(* Logix 5000 project; controller Machine_Maintenance_Lab2 vendor 1 type 14 code 155 rev 36.11; software revision 36.00 *)

TASK MainTask (continuous, watchdog 500 ms) : MainProgram

MODULES
   Local : vendor 1 type 14 code 155 (PointIO 0, rev 36.11)
      Discrete_IO : Embedded (PointIO 1, rev 36.11, Output RPI 20 ms)
END_MODULES

PROGRAM MainProgram   (* main routine TrafficLight *)
VAR
   Clock : FBD_TIMER := (PRE := 1000);
   ClockDone_NSGEWR : BOOL;
   ClockDone_NSREWG : BOOL;
   ClockDone_NSREWY : BOOL;
   ClockDone_NSYEWR : BOOL;
   counter : COUNTER := (PRE := 5);
   CycleCounter : COUNTER := (PRE := 5);
   delay : TIMER := (PRE := 10);
   EmerDone : BOOL;
   Emergency : BOOL;
   HighCycleTimer : COUNTER := (PRE := 700);
   i_CycleDone : ALIAS FOR o_CycleDone;
   i_GreenPB : ALIAS FOR Local:1:I.Data.0;
   i_GreenPB_ConveyorStart : ALIAS FOR i_GreenPB;
   i_GreenPBLight_Conveyor1ON : ALIAS FOR o_GreenPBLight_Conveyor1ON;
   i_NightModeButton : ALIAS FOR Local:1:I.Data.3;
   i_Pause : ALIAS FOR Pause;
   i_Piston : ALIAS FOR Local:1:O.Data.2;
   i_RedPB_StopButton : ALIAS FOR Local:1:I.Data.1;
   i_RedPBLight_Conveyor2ON : ALIAS FOR o_RedPBLight_Conveyor2ON;
   i_Turnkey : ALIAS FOR Local:1:I.Data.2;
   i_Turnkey_ItemSensor : ALIAS FOR i_Turnkey;
   ItemCounter1 : COUNTER := (PRE := 5);
   ItemCounterLeft : COUNTER := (PRE := 5);
   ItemCounterRight : COUNTER := (PRE := 6);
   LowCycleTimer : COUNTER := (PRE := 300);
   MaxState : DINT;
   myClock : FBD_TIMER;
   NewCycle : BOOL;
   NightMode : BOOL;
   o_CycleDone : BOOL;
   o_EWG : ALIAS FOR Local:1:O.Data.15;
   o_EWR : ALIAS FOR Local:1:O.Data.13;
   o_EWY : ALIAS FOR Local:1:O.Data.14;
   o_GreenPBLight : ALIAS FOR Local:1:O.Data.0;
   o_GreenPBLight_Conveyor1ON : ALIAS FOR o_GreenPBLight;
   o_NSG : ALIAS FOR Local:1:O.Data.7;
   o_NSR : ALIAS FOR Local:1:O.Data.5;
   o_NSY : ALIAS FOR Local:1:O.Data.6;
   o_Piston : ALIAS FOR i_Piston;
   o_RedPBLight : ALIAS FOR Local:1:O.Data.1;
   o_RedPBLight_Conveyor2ON : ALIAS FOR o_RedPBLight;
   OS_Out : BOOL;
   Pause : BOOL;
   preStart : DINT;
   resetBit : BOOL;
   ResetDelay : TIMER := (PRE := 500);
   Start : BOOL;
   StateCounter : FBD_COUNTER;
   ThreeSecTimer : TIMER := (PRE := 3000);
   timer : TIMER := (PRE := 5000);
   timerDoneLatch : BOOL;
   TimerHighCycle : TIMER := (PRE := 700);
   TimerLowCycle : TIMER := (PRE := 300);
   timerMem : BOOL;
   timerState : DINT;
   TurnkeyOneShot : BOOL := 1;
END_VAR

ROUTINE TrafficLight   (* structured text *)
   
   RTOR(myClock);
   
   // Set clock preset
   if(s:fs) then
   	myClock.PRE := 1000;
   	StateCounter.ACC := -1;
   end_if;
   
   // Pause button
   if ((not i_RedPB_StopButton)) then
   	Pause := 1;
   	Start := 0;
   end_if;
   
   // Start button
   if (i_GreenPB) then
   	Start := 1;
   	Pause := 0;
   end_if;
   
   // Timer enable
   if Start and (not i_Turnkey) then
   	myClock.Reset := 0;
   	myClock.TimerEnable := 1;
   	myClock.PRE := 1000;
   else
   	myClock.TimerEnable := 0;
   end_if;
   
   
   if myClock.DN then
   	StateCounter.ACC := StateCounter.ACC + 1;
   	myClock.Reset := 1;
   end_if;
   
   
   // Reset based on MaxState
   if (StateCounter.ACC > MaxState) then
   	StateCounter.ACC := 0;
   end_if;
   
   // Adjust state number to 8 if in night mode and change MaxState to 11
   if (i_NightModeButton) then
   	if (StateCounter.ACC < 8) then
   		StateCounter.ACC := 8;
   	end_if;
   
   	MaxState := 11;
   else
   
   	MaxState := 7;
   end_if;
   
   
   // Exit night mode reset
   if ((not i_NightModeButton) and (StateCounter.ACC >= 8)) then
   	StateCounter.ACC := 0;
   end_if;
   
   // Run through normal cycle or night mode if not EMER
   if (StateCounter.ACC = 0 or StateCounter.ACC = 1 or StateCounter.ACC = 2 or StateCounter.ACC = 3 or i_Turnkey) then
   	o_NSR := 1;
   else
   	o_NSR := 0;
   end_if;
   if ((StateCounter.ACC = 7 or StateCounter.ACC = 8 or StateCounter.ACC = 9) and (not i_Turnkey)) then
   	o_NSY := 1;
   else
   	o_NSY := 0;
   end_if;
   if ((StateCounter.ACC = 4 or StateCounter.ACC = 5 or StateCounter.ACC = 6) and (not i_Turnkey)) then
   	o_NSG := 1;
   else
   	o_NSG := 0;
   end_if;
   if (StateCounter.ACC = 4 or StateCounter.ACC = 5 or StateCounter.ACC = 6 or StateCounter.ACC = 7 or StateCounter.ACC = 10 or StateCounter.ACC = 11 or i_Turnkey) then
   	o_EWR := 1;
   else
   	o_EWR := 0;
   end_if;
   if (StateCounter.ACC = 3 and (not i_Turnkey)) then
   	o_EWY := 1;
   else
   	o_EWY := 0;
   end_if;
   if ((StateCounter.ACC = 0 or StateCounter.ACC = 1 or StateCounter.ACC = 2) and (not i_Turnkey)) then
   	o_EWG := 1;
   else
   	o_EWG := 0;
   end_if;
END_ROUTINE
END_PROGRAM
